INTERFACE I_Lift EXTENDS I_Position

PROPERTY Assigned : BOOL
GET
END_GET
SET
END_SET
END_PROPERTY

METHOD Call : HRESULT
VAR_INPUT
	Position : LREAL;
	Velocity : LREAL;
END_VAR
END_METHOD

END_INTERFACE

(* stored: Version 1.1.0.1
   Itf I_Lift: Id {aabca9f0-6a1e-4b18-a681-bf2d8e7e4273}
   Property Assigned: Id {5bc2abc7-8576-41cd-b6d7-7345a20b1674}
   Get Get: Id {f36b38f8-2fd2-4947-8c11-9e282d764737}
   Set Set: Id {641fd3e2-af31-4d87-8fee-210dc813ce4a}
   Method Call: Id {2883bae7-2d85-4d90-bea8-3c456db1f029} *)
